FUNCTION_BLOCK VECTOR_CROSS_P (* Cross product between two vector *)
  (* Standard: 61499-2 *)
  (* Version 1.0, 02-05-12, GASR, Universidade do Estado de Santa Catarina *)
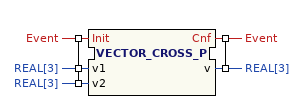
  EVENT_INPUT
    Init WITH v1, v2;
  END_EVENT
  EVENT_OUTPUT
    Cnf WITH v;
  END_EVENT
  VAR_INPUT
    v1 : ARRAY [0..2] OF REAL;
    v2 : ARRAY [0..2] OF REAL;
  END_VAR
  VAR_OUTPUT
    v : ARRAY [0..2] OF REAL;
  END_VAR
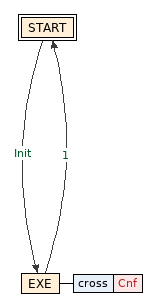
  EC_STATES
    START;
    EXE : cross -> Cnf;
  END_STATES
  EC_TRANSITIONS
    START TO EXE := Init;
    EXE TO START := 1;
  END_TRANSITIONS
  ALGORITHM cross IN Lua:
v[1] = ((v1[2]*v2[3]) - (v2[2]*v1[3]))
v[2] = ((v1[3]*v2[1]) - (v2[3]*v1[1]))
v[3] = ((v1[1]*v2[2]) - (v2[1]*v1[2]))
  END_ALGORITHM
END_FUNCTION_BLOCK
